TYPE ST_Chart :
STRUCT
        Distance : REAL;
        Force    : REAL;
END_STRUCT
END_TYPE

(* stored: Version 1.1.0.1, ProductVersion 3.1.4024.12
   DUT ST_Chart: Id {e16c24a0-2f05-4910-b5bc-d65b1ffeb27b} *)
